{attribute 'pack_mode' := '2'}
TYPE ST_MOVER_CTRL :
STRUCT
  Cmd             : E_MOVER_CTRL;  // order to execute on mover
END_STRUCT
END_TYPE

(* stored: Version 1.1.0.1, ProductVersion 3.1.4024.12
   DUT ST_MOVER_CTRL: Id {47f81db5-ead7-447a-86d8-5557b98eebc2} *)
